FUNCTION GetIndexOfAxisId : uint
VAR_INPUT
  nAxisId   : UDINT;
END_VAR
VAR
  _idx,
  _ret      : UINT;
END_VAR


FOR _idx := 1 TO PLC_CONSTANT.MAX_AXIS
DO
  IF (GVL_AXIS.AxisRef[_idx].NcToPlc.AxisId = nAxisId)
  THEN
    _ret  := _idx;
    EXIT;
  END_IF
END_FOR

GetIndexOfAxisId  := _ret;

END_FUNCTION

(* stored: Version 1.1.0.1, ProductVersion 3.1.4024.12
   POU GetIndexOfAxisId: Id {076f32c0-9c5a-08b8-1caa-b76ab51c5c08}, SpecialFunc None *)
